{attribute 'linkalways'} 
{attribute 'no_explicit_call' := 'This FB is a CLASS and must be accessed using methods or properties'}
{attribute 'enable_dynamic_creation'}
FUNCTION_BLOCK Node_F_VN_FillRectangle EXTENDS VisionNode
VAR
    nTopLeftX : _UDINT(0);
    nTopLeftY : _UDINT(0);
    nBottomRightX : _UDINT(0);
    nBottomRightY : _UDINT(0);
    ipDestImage : _ITcVnImage;
    aColor : _TcVnVector4_LREAL;
    hrPrev : _HRESULT(S_OK);
	hresult : _HRESULT(S_OK);
END_VAR

METHOD PUBLIC  Clone : I_Node
VAR
	pNode : POINTER TO Node_F_VN_FillRectangle;
END_VAR
pNode := __NEW(Node_F_VN_FillRectangle);
Clone := pNode^;
END_METHOD

METHOD FB_init : BOOL
VAR_INPUT
	bInitRetains : BOOL; // if TRUE, the retain variables are initialized (warm start / cold start)
	bInCopyCode : BOOL;  // if TRUE, the instance afterwards gets moved into the copy code (online change)
END_VAR
AddParameter('nTopLeftX', nTopLeftX);
AddParameter('nTopLeftY', nTopLeftY);
AddParameter('nBottomRightX', nBottomRightX);
AddParameter('nBottomRightY', nBottomRightY);
AddInput('ipDestImage', ipDestImage);
AddInput('aColor', aColor);
AddInput('hrPrev', hrPrev);
AddOutput('ipDestImage', ipDestImage);
AddOutput('hresult',hresult);
END_METHOD

METHOD PROTECTED OnExecute
hresult.Value := F_VN_FillRectangle(
    nTopLeftX := nTopLeftX.Value,
    nTopLeftY := nTopLeftY.Value,
    nBottomRightX := nBottomRightX.Value,
    nBottomRightY := nBottomRightY.Value,
	ipDestImage := ipDestImage.Value,
    aColor := aColor.Value,
	hrPrev:= hrPrev.Value);
END_METHOD

METHOD PUBLIC PreExecutionCheck
VAR_INPUT
	Check : I_PreExecutionChecks;
END_VAR
Check.IsTrue(ipDestImage.IsValid, 'ipDestImage must contain an image');
END_METHOD

END_FUNCTION_BLOCK

(* stored: Version 1.1.0.1, ProductVersion 3.1.4024.13
   POU Node_F_VN_FillRectangle: Id {1b439b58-df0a-0f2b-2bf2-894d6a66240c}, SpecialFunc None
   Folder Constructor: Id {936fb44b-5a2e-06e7-1acd-e4c6ef16c94b}
   Method Clone: Id {9224ce0a-eea1-032c-2dc6-de836facf5ca}
   Method FB_init: Id {ea6781a2-fe14-0836-2ebd-e3d6ae3a8689}
   Method OnExecute: Id {e41f2a75-4907-04b1-35c9-5e013813a3fc}
   Method PreExecutionCheck: Id {27971d06-658d-0edf-2639-ac93f3081e71} *)
